// TIA Portal project "单按钮控制两台电机互启互停" (V15.1)

(* hardware
DEVICE "S7-1200 station_1"  S7-1200 Station
   slot 0: "Rack_0"  S7-1200 Rack  Rack  V1.0
   slot 1: "PLC_1"  CPU 1212C DC/DC/DC  6ES7 212-1AE40-0XB0  V4.2
DEVICE "HMI_1"  KTP700 Basic PN Portrait
   slot 0: "HMI_1"  KTP700 Basic PN Portrait  6AV2 123-2GB03-0AX0  15.1.0.0
   slot 1: "HMI_RT_1"  KTP700 Basic PN Portrait  6AV2 123-2GB03-0AX0  15.1.0.0
   slot 5: "HMI_1.IE_CP_1"  PROFINET Interface  15.0.1.0
      slot 1: "PROFINET Interface_1"  PROFINET Interface
         slot 1: "Port_1"  Port
*)

// ===== PLC "PLC_1"  CPU 1212C DC/DC/DC =====

VAR_GLOBAL   // PLC tag table "默认变量表"
   "Tag_1" AT %M10.0 : Bool;
END_VAR

VAR_GLOBAL   // PLC tag table "io2"
   "开启" AT %I0.4 : Bool;
   "中间标志1" AT %M1.0 : Bool;
   "中间标志2" AT %M1.1 : Bool;
   "电机1" AT %Q0.4 : Bool;
   "电机2" AT %Q0.5 : Bool;
   "中间标志3" AT %M1.2 : Bool;
END_VAR

VAR_GLOBAL   // PLC tag table "io1"
   "启动" AT %I0.0 : Bool;
   "停止" AT %I0.1 : Bool;
   "中间" AT %M0.0 : Bool;
   "中间1" AT %M0.1 : Bool;
   "电机" AT %Q0.0 : Bool;
END_VAR

ORGANIZATION_BLOCK "Main"   // OB1, LAD, ProgramCycle
TITLE = "Main Program Sweep (Cycle)"
{ S7_Optimized_Access := 'TRUE' }
VERSION : 0.1
   VAR_INPUT
      Initial_Call : Bool;   // Initial call of this OB
      Remanence : Bool;   // =True, if remanent data are available
   END_VAR
   VAR_TEMP   // added for the SCL form of the ladder/FBD networks
      _w1 : Bool;
      _w2 : Bool;
      _w3 : Bool;
   END_VAR
BEGIN

REGION Network 1
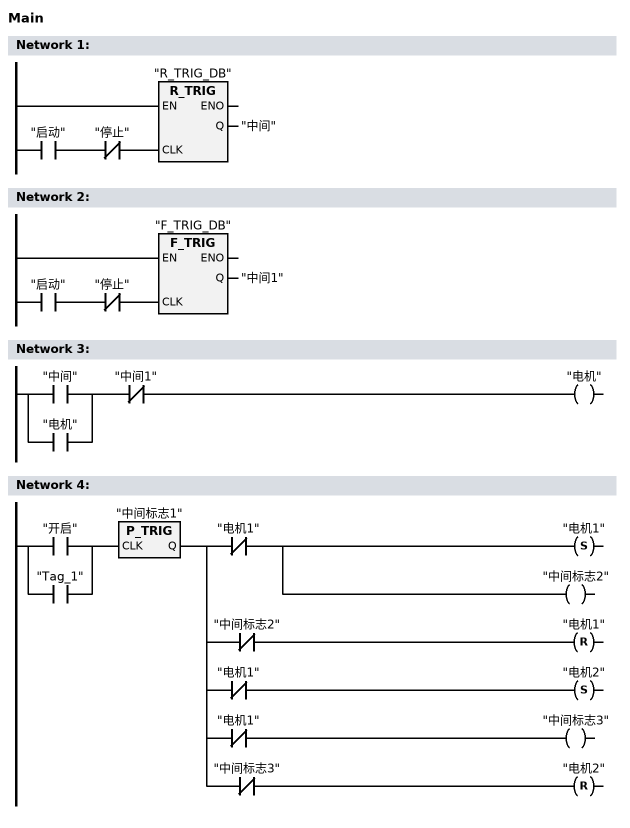
   "R_TRIG_DB"(CLK := "启动" AND NOT "停止", Q => "中间");   // R_TRIG
END_REGION

REGION Network 2
   "F_TRIG_DB"(CLK := "启动" AND NOT "停止", Q => "中间1");   // F_TRIG
END_REGION

REGION Network 3
   RUNG wire#powerrail
      Contact( "中间" )
      wire#w1
      I_Contact( "中间1" )
      Coil( "电机" )
   END_RUNG
   RUNG wire#powerrail
      Contact( "电机" )
   END_RUNG wire#w1
   // the same network as SCL:
   "电机" := ("中间" OR "电机") AND NOT "中间1";
END_REGION

REGION Network 4
   RUNG wire#powerrail
      Contact( "开启" )
      wire#w1
      P_Trig( "中间标志1" )
      wire#w2
      I_Contact( "电机1" )
      wire#w3
      S_Coil( "电机1" )
   END_RUNG
   RUNG wire#powerrail
      Contact( "Tag_1" )
   END_RUNG wire#w1
   RUNG wire#w3
      Coil( "中间标志2" )
   END_RUNG
   RUNG wire#w2
      I_Contact( "中间标志2" )
      R_Coil( "电机1" )
   END_RUNG
   RUNG wire#w2
      I_Contact( "电机1" )
      S_Coil( "电机2" )
   END_RUNG
   RUNG wire#w2
      I_Contact( "电机1" )
      Coil( "中间标志3" )
   END_RUNG
   RUNG wire#w2
      I_Contact( "中间标志3" )
      R_Coil( "电机2" )
   END_RUNG
   // the same network as SCL:
   #_w1 := "开启" OR "Tag_1";
   #_w2 := #_w1 AND NOT "中间标志1";   // rising edge
   "中间标志1" := #_w1;
   #_w3 := #_w2 AND NOT "电机1";
   IF #_w3 THEN "电机1" := TRUE; END_IF;
   "中间标志2" := #_w3;
   IF #_w2 AND NOT "中间标志2" THEN "电机1" := FALSE; END_IF;
   IF #_w2 AND NOT "电机1" THEN "电机2" := TRUE; END_IF;
   "中间标志3" := #_w2 AND NOT "电机1";
   IF #_w2 AND NOT "中间标志3" THEN "电机2" := FALSE; END_IF;
END_REGION
END_ORGANIZATION_BLOCK

(* ===== HMI "HMI_RT_1" =====
system functions are stored by id; their names below are inferred from use
connection "HMI_连接_1": ETHERNET, SMART_S7_1200_OMS

HMI tags "默认变量表"
   "Tag_ScreenNumber" : UInt, internal
   "Tag_1" : Bool = PLC Tag_1 AT %M10.0, 1 s
   "电机1" : Bool = PLC 电机1 AT %Q0.4, 1 s
   "电机2" : Bool = PLC 电机2 AT %Q0.5, 1 s

Template "模板_1" 480x800
   Button "起始画面" at 428,61 size 50x71; TextOff '起始画面'; PictureOff "NavigateHome_KTP700_Basic_PN_Portrait_TR"; PictureOn "NavigateHome_KTP700_Basic_PN_Portrait_TR"
      on Release: ActivateScreen("根画面", 0)
   Button "Template_Button" at 428,172 size 50x71; TextOff 'Text'
   Button "Template_Button_1" at 428,283 size 50x71; TextOff 'Text'
   Button "Template_Button_2" at 428,394 size 50x71; TextOff 'Text'
   Button "Template_Button_3" at 428,505 size 50x71; TextOff 'Text'
   Button "Template_Button_4" at 428,616 size 50x71; TextOff 'Text'
   Button "退出" at 428,727 size 50x71; TextOff '退出'; PictureOff "ExitRuntime_KTP700_Basic_PN_Portrait_TR"; PictureOn "ExitRuntime_KTP700_Basic_PN_Portrait_TR"
      on Release: StopRuntime(0)
   SymbolicIOField "Symbolic_IO_Field_Screen" at 109,11 size 264x38; TextOff '0'; TextOn '1'; TextList "TextList_ScreenNames"
      ProcessValue <- "Tag_ScreenNumber"
      on Change: ActivateScreenByNumber("Tag_ScreenNumber", 0)
   DateTimeField "HmiScreenItemData" at 375,30 size 105x30
   DateTimeField "HmiScreenItemData_1" at 375,0 size 105x30
   GraphicView "Logo" at 0,0 size 107x60; Picture "HMI_1 的 Logo"

screen "根画面" 480x800, template "模板_1"
   on GenerateScreen: SetTag("Tag_ScreenNumber", 1)
   TextField "HmiScreenItemData" at 43,404 size 343x46; Text '欢迎进入 HMI_1 (KTP700 Basic+ PN Portrait)！'
   Button "按钮_1" at 43,164 size 96x32; TextOff '开启'
      on Press: SetBit("Tag_1")
      on Release: ResetBit("Tag_1")
   Circle "圆_1" at 220,157 size 48x48
      Appearance <- "电机1"
   Circle "圆_2" at 331,162 size 48x48
      Appearance <- "电机2"
   TextField "文本域_1" at 220,239 size 48x20; Text '电机1'
   TextField "文本域_2" at 331,239 size 48x20; Text '电机2'
*)